// TIA Portal V19 export
TYPE "LAF_typeAxisDiagValues"
TITLE = LAF_typeAxisDiagValues
// Setpoint and actual values of a Technology Object
// stored: Access Published
   STRUCT
      position { ExternalWritable := 'False'} : LReal;   // Position setpoint
      velocity { ExternalWritable := 'False'} : LReal;   // Velocity setpoint / speed setpoint
      actualPosition { ExternalWritable := 'False'} : LReal;   // Actual position
      actualVelocity { ExternalWritable := 'False'} : LReal;   // Actual velocity
      actualSpeed { ExternalWritable := 'False'} : LReal;   // PROFIdrive drive = actual speed of the motor / drive with analog setpoint = 0.0 / drives with linear motor = 0.0
   END_STRUCT;
END_TYPE
